RoboDK station: Stringer B-Bot-BOX2.rdk

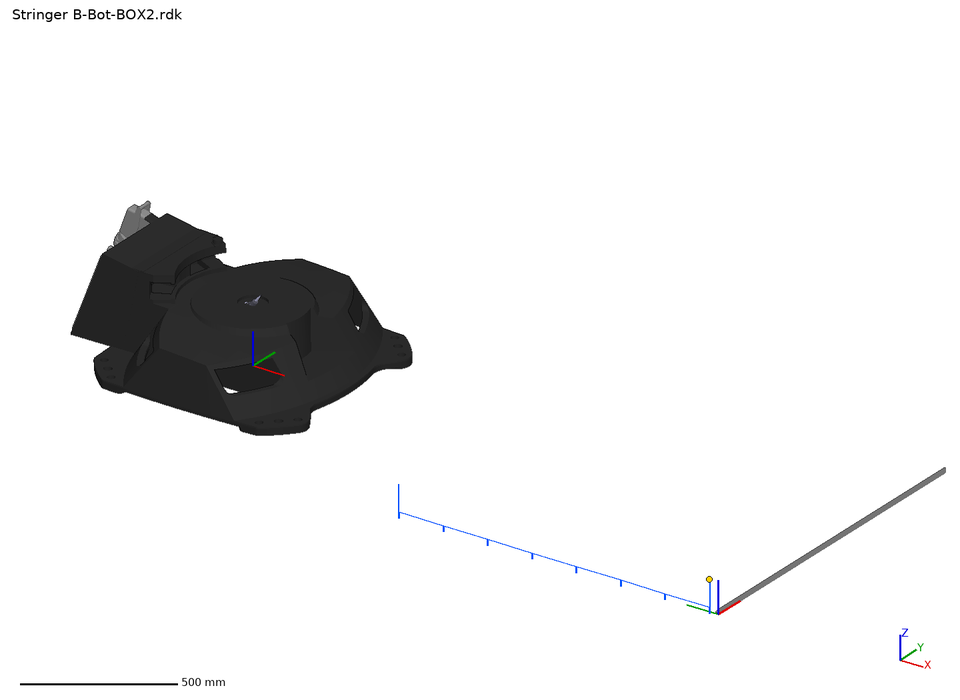
[picture v0: the station drawn from its stored meshes, robots at their saved joint values, targets as dots, program paths as lines]
Station Stringer B-Bot-BOX2 (saved by RoboDK 5.2.3). Poses are relative to the parent item; angles as X-Y-Z fixed-axis rotations.
  - frame KUKA KR 210 R2700 extra Base at (0, 0, 0) mm
    - robot KUKA KR 210 R2700 extra: 6 axes, payload 210 kg, reach 2696 mm, repeatability 0.06 mm, weight 1068 kg
        joint limits [-185, -140, -120, -350, -125, -350] to [185, -5, 155, 350, 125, 350]; home [0, -90, 90, 0, 0, 0]; saved at [-39.004, -26.693, 86.216, 93.944, 23.392, -126.483]
      - tool Spindle, TCP at (32, 0, 260) mm, rotated rx 0 ry 39 rz 0 deg, size 157.3 x 72 x 259.9 mm
  - frame Frame 2 at (1800, 0, -372.68) mm, rotated rx 0 ry 0 rz 90 deg
    - object L-Stringer B-Bot-BOX2 at (0, 0, 0) mm, size 1250 x 20 x 20 mm, geometry from L-Stringer B-Bot-BOX2.stl
    - object Stringer B-Bot-BOX2 at (0, 0, 0) mm, rotated rx 0 ry 0 rz -90 deg, 8 curves, geometry from Point 8
  - machining project Point settings: rotZ(0) | rotX(0)*rotY(0) | rotz(0) | onStart | onPathStart | onApproach | onPoint | onRetract | onFinish | SetRPM(%1) | SetTool(%1) | Extruder(%1) | default | default | OutOnMov(%1) | OutOffMov(%1) | onPathFinish | M_RunCode(%1) | riverData=C:\Windows\System32\Driv | PS_BROWSER_APP_PROFILE_STRING=Inter | PS_BROWSER_USER_PROFILE_STRING=Defa | OCALAPPDATA=C:\Users\jbert\AppData\Loc | OneDrive=C:\Users\jbert\O | Path=C:\Program Files (x86)\NVIDIA Corpora
  - program Point (51 instructions, listed below)
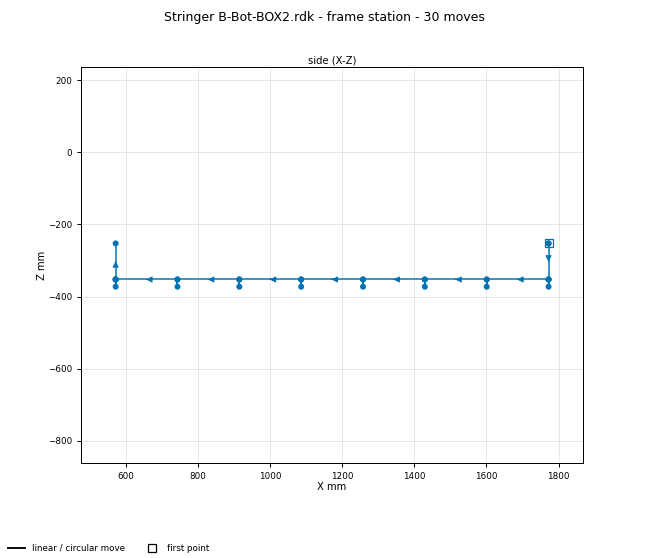
[picture p0: tool path of Stringer B-Bot-BOX2.rdk in frame station, 30 of 30 moves have a stored position in this frame; points joined in program order, loops and branches not executed]

--- program Point (robot KUKA KR 210 R2700 extra) ---
  Smooth(1)
  Set speed (1000.0 mm/s)
  Set Ref.: Frame 2
  Set Tool: Spindle
  Show Spindle
  MoveJ 1 to (-10.01, 27.74, 120) mm, rotated rx 180 ry 0 rz 180 deg; joints [-1.048, -34.012, 111.841, 178.538, 26.831, -179.51]
  MoveL 2 to (-10.01, 27.74, 120) mm, rotated rx 180 ry 0 rz 180 deg; joints [-1.048, -34.012, 111.841, 178.538, 26.831, -179.51]
  MoveL 3 to (-10.01, 27.74, 20) mm, rotated rx -180 ry 0 rz -180 deg; joints [-1.048, -28.683, 109.198, 178.661, 29.517, -179.649]
  MoveL 4 to (-10.01, 27.74, 20) mm, rotated rx -180 ry 0 rz -180 deg; joints [-1.048, -28.683, 109.198, 178.661, 29.517, -179.649]
  Set speed (50.0 mm/s)
  MoveL 5 to (-10.01, 27.74, 0) mm, rotated rx 180 ry 0 rz -180 deg; joints [-1.048, -27.625, 108.622, 178.68, 29.999, -179.672]
  MoveL 6 to (-10.01, 27.74, 20) mm, rotated rx -180 ry 0 rz -180 deg; joints [-1.048, -28.683, 109.198, 178.661, 29.517, -179.649]
  Set speed (1000.0 mm/s)
  MoveL 7 to (-10.01, 199.17, 20) mm, rotated rx 180 ry 0 rz 180 deg; joints [-7.485, -28.59, 108.533, 170.281, 29.054, -177.315]
  Set speed (50.0 mm/s)
  MoveL 8 to (-10.01, 199.17, 0) mm, rotated rx 180 ry 0 rz 180 deg; joints [-7.485, -27.538, 107.96, 170.424, 29.525, -177.479]
  MoveL 9 to (-10.01, 199.17, 20) mm, rotated rx 180 ry 0 rz 180 deg; joints [-7.485, -28.59, 108.533, 170.281, 29.054, -177.315]
  Set speed (1000.0 mm/s)
  MoveL 10 to (-10.01, 370.6, 20) mm, rotated rx -180 ry 0 rz -180 deg; joints [-13.738, -28.334, 106.869, 161.422, 27.975, -174.224]
  Set speed (50.0 mm/s)
  MoveL 11 to (-10.01, 370.6, 0) mm, rotated rx 180 ry 0 rz 180 deg; joints [-13.738, -27.297, 106.301, 161.699, 28.42, -174.539]
  MoveL 12 to (-10.01, 370.6, 20) mm, rotated rx -180 ry 0 rz -180 deg; joints [-13.738, -28.334, 106.869, 161.422, 27.975, -174.224]
  Set speed (1000.0 mm/s)
  MoveL 13 to (-10.01, 542.03, 20) mm, rotated rx -180 ry 0 rz -180 deg; joints [-19.675, -27.86, 104.216, 151.641, 26.492, -169.745]
  Set speed (50.0 mm/s)
  MoveL 14 to (-10.01, 542.03, 0) mm, rotated rx -180 ry 0 rz -180 deg; joints [-19.675, -26.845, 103.657, 152.069, 26.894, -170.223]
  MoveL 15 to (-10.01, 542.03, 20) mm, rotated rx -180 ry 0 rz -180 deg; joints [-19.675, -27.86, 104.216, 151.641, 26.492, -169.745]
  Set speed (1000.0 mm/s)
  MoveL 16 to (-10.01, 713.46, 20) mm, rotated rx 180 ry 0 rz 180 deg; joints [-25.204, -27.095, 100.589, 140.503, 24.919, -163.312]
  Set speed (50.0 mm/s)
  MoveL 17 to (-10.01, 713.46, 0) mm, rotated rx 180 ry 0 rz 180 deg; joints [-25.204, -26.107, 100.038, 141.094, 25.258, -163.964]
  MoveL 18 to (-10.01, 713.46, 20) mm, rotated rx 180 ry 0 rz 180 deg; joints [-25.204, -27.095, 100.589, 140.503, 24.919, -163.312]
  Set speed (1000.0 mm/s)
  MoveL 19 to (-10.01, 884.89, 20) mm, rotated rx 180 ry 0 rz 180 deg; joints [-30.273, -25.962, 95.989, 127.718, 23.645, -154.574]
  Set speed (50.0 mm/s)
  MoveL 20 to (-10.01, 884.89, 0) mm, rotated rx 180 ry 0 rz 180 deg; joints [-30.273, -25.004, 95.446, 128.458, 23.9, -155.383]
  MoveL 21 to (-10.01, 884.89, 20) mm, rotated rx 180 ry 0 rz 180 deg; joints [-30.273, -25.962, 95.989, 127.718, 23.645, -154.574]
  Set speed (1000.0 mm/s)
  MoveL 22 to (-10.01, 1056.32, 20) mm, rotated rx -180 ry 0 rz -180 deg; joints [-34.869, -24.38, 90.401, 113.434, 23.087, -143.665]
  Set speed (50.0 mm/s)
  MoveL 23 to (-10.01, 1056.32, 0) mm, rotated rx 180 ry 0 rz 180 deg; joints [-34.869, -23.454, 89.863, 114.261, 23.244, -144.565]
  MoveL 24 to (-10.01, 1056.32, 20) mm, rotated rx -180 ry 0 rz -180 deg; joints [-34.869, -24.38, 90.401, 113.434, 23.087, -143.665]
  Set speed (1000.0 mm/s)
  MoveL 25 to (-10.01, 1227.74, 20) mm, rotated rx 180 ry 0 rz 180 deg; joints [-39.004, -22.268, 83.771, 98.474, 23.606, -131.421]
  Set speed (50.0 mm/s)
  MoveL 26 to (-10.01, 1227.74, 0) mm, rotated rx 180 ry 0 rz -180 deg; joints [-39.004, -21.372, 83.231, 99.277, 23.661, -132.298]
  MoveL 27 to (-10.01, 1227.74, 20) mm, rotated rx 180 ry 0 rz 180 deg; joints [-39.004, -22.268, 83.771, 98.474, 23.606, -131.421]
  MoveL 28 to (-10.01, 1227.74, 20) mm, rotated rx 180 ry 0 rz 180 deg; joints [-39.004, -22.268, 83.771, 98.474, 23.606, -131.421]
  Set speed (1000.0 mm/s)
  MoveL 29 to (-10.01, 1227.74, 20) mm, rotated rx 180 ry 0 rz 180 deg; joints [-39.004, -22.268, 83.771, 98.474, 23.606, -131.421]
  MoveL 30 to (-10.01, 1227.74, 120) mm, rotated rx 180 ry 0 rz -180 deg; joints [-39.004, -26.693, 86.216, 93.944, 23.392, -126.483]
